FUNCTION Buffer_Layout_Set_Bool_Array : UINT
VAR_INPUT
	Amount : UINT;
END_VAR

VAR_IN_OUT
	Layout : Buffer_Layout;
END_VAR

VAR
END_VAR

END_FUNCTION

(* stored: Version 1.1.0.1, ProductVersion 3.1.4024.10
   POU Buffer_Layout_Set_Bool_Array: Id {64170c66-22af-4c41-a639-133b67fc81cb}, SpecialFunc None *)
